  Script: wp_InsBat2Ret[2] = wp_InsBat2Ret[2] - 0.10
  MoveL speed 250 mm/s, acceleration 1200 mm/s^2 (useActiveTCP=true) feature=Fearure_2_2P_Of
    Waypoint Waypoint (Variable): variable=wp_InsBat2Ret
  URCap Gripper (Robotiq_Grippers, Robotiq Inc.) dataModel(position=100.0, force=0.0, speed=100.0, positionInDouble=100.0, forceInDouble=0.0, speedInDouble=100.0, slaveIds=[9], blocking=true)
SubProgram ExtractCoinBattery (keepSynchronizedWithDisk=false)
  wp_CoinBatApp := wp_origin
  Script: wp_CoinBatApp[0] = -0.0328
  Script: wp_CoinBatApp[1] = 0.1238 + 0.002
  Script: wp_CoinBatApp[2] = 0.07
  MoveL speed 250 mm/s, acceleration 1200 mm/s^2 (useActiveTCP=true) feature=Fearure_2_2P_Of
    Waypoint Waypoint (Variable): variable=wp_CoinBatApp
  wp_CoinBatExt := wp_CoinBatApp
  Script: wp_CoinBatExt[2] = 0.115
  MoveL speed 250 mm/s, acceleration 1200 mm/s^2 (useActiveTCP=true) feature=Fearure_2_2P_Of
    Waypoint Waypoint (Variable): variable=wp_CoinBatExt
  URCap Find Surface (Robotiq_Copilot, Robotiq Inc.) dataModel(NodeInitializedKey=true, WaitForSteadyWrenchOptionKey=false, ZeroSensorBeforeKey=true, ls_distance=20.0, ls_direction=X-, ls_if_distance=false, ls_if_force=false, ls_force=35.0, ls_speed=5.0); state(isChildrenLocked=true)
    'Add Stop conditions from the Find Surface node'
  Wait NoWait
  Script: wp_CoinBatExt[2] = 0.07
  MoveL speed 250 mm/s, acceleration 1200 mm/s^2 (useActiveTCP=true) feature=Fearure_2_2P_Of
    Waypoint Waypoint (Variable): variable=wp_CoinBatExt
  SuppressedNode
    Script: wp_CoinBatExt[1] = wp_CoinBatExt[1] + 0.1238
  SuppressedNode
    Script: wp_CoinBatExt[3] = 0.785398
SubProgram ReleaseTool (keepSynchronizedWithDisk=false)
  wp_RelToolApp := wp_origin
  Script: wp_RelToolApp[0] = -0.0328
  Script: wp_RelToolApp[1] = 0.18
  Script: wp_RelToolApp[2] = 0.07
  MoveL speed 250 mm/s, acceleration 1200 mm/s^2 (useActiveTCP=true) feature=Fearure_2_2P_Of
    Waypoint Waypoint (Variable): variable=wp_RelToolApp
  URCap Gripper (Robotiq_Grippers, Robotiq Inc.) dataModel(position=50.0, force=0.0, speed=100.0, positionInDouble=50.0, forceInDouble=0.0, speedInDouble=100.0, slaveIds=[9], blocking=true)
  Script: wp_RelToolApp[2] = 0
  MoveL speed 250 mm/s, acceleration 1200 mm/s^2 (useActiveTCP=true) feature=Fearure_2_2P_Of
    Waypoint Waypoint (Variable): variable=wp_RelToolApp
  URCap Gripper (Robotiq_Grippers, Robotiq Inc.) dataModel(position=100.0, force=0.0, speed=100.0, positionInDouble=100.0, forceInDouble=0.0, speedInDouble=100.0, slaveIds=[9], blocking=true)
SubProgram PickPlaceCoinBattery (keepSynchronizedWithDisk=false)
  URCap Gripper (Robotiq_Grippers, Robotiq Inc.) dataModel(position=50.0, force=0.0, speed=100.0, positionInDouble=50.0, forceInDouble=0.0, speedInDouble=100.0, slaveIds=[9], blocking=true)
  wp_PickCoinApp := wp_origin
  Script: wp_PickCoinApp[0] = -0.0328
  Script: wp_PickCoinApp[1] = 0.1238
  Script: wp_PickCoinApp[2] = 0.14
  Script: wp_PickCoinApp[5] = d2r(90)
  MoveL speed 250 mm/s, acceleration 1200 mm/s^2 (useActiveTCP=true) feature=Fearure_2_2P_Of
    Waypoint Waypoint (Variable): variable=wp_PickCoinApp
  URCap Gripper (Robotiq_Grippers, Robotiq Inc.) dataModel(position=100.0, force=0.0, speed=0.0, positionInDouble=100.0, forceInDouble=0.0, speedInDouble=0.0, slaveIds=[9], blocking=true)
  Script: wp_PickCoinApp[2] = 0.12
  MoveL speed 250 mm/s, acceleration 1200 mm/s^2 (useActiveTCP=true) feature=Fearure_2_2P_Of
    Waypoint Waypoint (Variable): variable=wp_PickCoinApp
  Script: wp_PickCoinApp[1] = 0.09
  MoveL speed 250 mm/s, acceleration 1200 mm/s^2 (useActiveTCP=true) feature=Fearure_2_2P_Of
    Waypoint Waypoint (Variable): variable=wp_PickCoinApp
  Script: wp_PickCoinApp[2] = 0.13
  MoveL speed 250 mm/s, acceleration 1200 mm/s^2 (useActiveTCP=true) feature=Fearure_2_2P_Of
    Waypoint Waypoint (Variable): variable=wp_PickCoinApp
  URCap Gripper (Robotiq_Grippers, Robotiq Inc.) dataModel(position=65.0, force=0.0, speed=0.0, positionInDouble=65.0, forceInDouble=0.0, speedInDouble=0.0, slaveIds=[9], blocking=true)
  Script: wp_PickCoinApp[2] = 0
  MoveL speed 250 mm/s, acceleration 1200 mm/s^2 (useActiveTCP=true) feature=Fearure_2_2P_Of
    Waypoint Waypoint (Variable): variable=wp_PickCoinApp
  URCap Gripper (Robotiq_Grippers, Robotiq Inc.) dataModel(position=100.0, force=0.0, speed=100.0, positionInDouble=100.0, forceInDouble=0.0, speedInDouble=100.0, slaveIds=[9], blocking=true)
SubProgram PressRedButton (keepSynchronizedWithDisk=false)
  wp_RedButApp := wp_origin
  Script: wp_RedButApp[0] = wp_RedButApp[0] - 0.0555
  Script: wp_RedButApp[1] = wp_RedButApp[1] + 0.03
  MoveL speed 250 mm/s, acceleration 1200 mm/s^2 (useActiveTCP=true) feature=Feature_1
    Waypoint Waypoint (Variable): variable=wp_RedButApp
  Popup Message (haltProgram=false inputType=Variable) variable=wp_RedButApp
  wp_RedButPress := wp_RedButApp
  Script: wp_RedButPress[2] = wp_RedButPress[2] + 0.125
  MoveL speed 250 mm/s, acceleration 1200 mm/s^2 (useActiveTCP=true) feature=Feature_1
    Waypoint Waypoint (Variable): variable=wp_RedButPress
  URCap Find Surface (Robotiq_Copilot, Robotiq Inc.) dataModel(NodeInitializedKey=true, WaitForSteadyWrenchOptionKey=false, ls_force=5.0, ls_speed=30.0, ls_distance=10.0, ls_if_distance=false, ls_if_force=true, ZeroSensorBeforeKey=true); state(isChildrenLocked=true)
    'Add Stop conditions from the Find Surface node'
    URCap If surface found (Robotiq_Copilot, Robotiq Inc.)
      'Sequence if force threshold is reached'
  wp_RedButRet := wp_RedButApp
  MoveL speed 250 mm/s, acceleration 1200 mm/s^2 (useActiveTCP=true) feature=Feature_1
    Waypoint Waypoint (Variable): variable=wp_RedButRet
